LIN {X 0,Y 107.526,Z 478.473,A -85,B 0,C 180,E1 -28773.988,E2 -28773.988} C_VEL
LIN {X 0,Y 117.989,Z 469.59,A -85,B 0,C 180,E1 -28777.405,E2 -28777.405} C_VEL
LIN {X 0,Y 127.771,Z 459.826,A -85,B 0,C 180,E1 -28780.218,E2 -28780.218} C_VEL
LIN {X 0,Y 128.984,Z 458.465,A -85,B 0,C 180,E1 -28780.541,E2 -28780.541} C_VEL
LIN {X 0,Y 129.571,Z 457.629,A -85,B 0,C 180,E1 -28781.007,E2 -28781.007} C_VEL
LIN {X 0,Y 130.543,Z 454.991,A -85,B 0,C 180,E1 -28784.384,E2 -28784.384} C_VEL
LIN {X 0,Y 131.123,Z 453.011,A -85,B 0,C 180,E1 -28787.62,E2 -28787.62} C_VEL
LIN {X 0,Y 131.637,Z 451.555,A -85,B 0,C 180,E1 -28790.783,E2 -28790.783} C_VEL
LIN {X 0,Y 132.063,Z 450.596,A -85,B 0,C 180,E1 -28793.89,E2 -28793.89} C_VEL
LIN {X 0,Y 132.436,Z 450.06,A -85,B 0,C 180,E1 -28796.958,E2 -28796.958} C_VEL
LIN {X 0,Y 132.765,Z 450.031,A -85,B 0,C 180,E1 -28800,E2 -28800} C_VEL
LIN {X 0,Y 132.291,Z 452.688,A -85,B 0,C 180,E1 -28806.099,E2 -28806.099} C_VEL
LIN {X 0,Y 132.117,Z 455.556,A -85,B 0,C 180,E1 -28810.73,E2 -28810.73} C_VEL
LIN {X 0,Y 131.781,Z 457.018,A -85,B 0,C 180,E1 -28812.317,E2 -28812.317} C_VEL
LIN {X 0,Y 130.688,Z 459.886,A -85,B 0,C 180,E1 -28814.539,E2 -28814.539} C_VEL
LIN {X 0,Y 128.33,Z 462.983,A -85,B 0,C 180,E1 -28815.54,E2 -28815.54} C_VEL
LIN {X 0,Y 124.785,Z 467.253,A -85,B 0,C 180,E1 -28816.775,E2 -28816.775} C_VEL
LIN {X 0,Y 115.231,Z 476.64,A -85,B 0,C 180,E1 -28819.031,E2 -28819.031} C_VEL
LIN {X 0,Y 104.384,Z 485.862,A -85,B 0,C 180,E1 -28822.218,E2 -28822.218} C_VEL
LIN {X 0,Y 94.042,Z 493.562,A -85,B 0,C 180,E1 -28826.263,E2 -28826.263} C_VEL
LIN {X 0,Y 82.992,Z 500.795,A -85,B 0,C 180,E1 -28832.133,E2 -28832.133} C_VEL
LIN {X 0,Y 73.155,Z 506.533,A -85,B 0,C 180,E1 -28839.777,E2 -28839.777} C_VEL
LIN {X 0,Y 64.941,Z 510.906,A -85,B 0,C 180,E1 -28849.511,E2 -28849.511} C_VEL
LIN {X 0,Y 59.141,Z 514.04,A -85,B 0,C 180,E1 -28861.62,E2 -28861.62} C_VEL
LIN {X 0,Y 56.399,Z 515.993,A -85,B 0,C 180,E1 -28875.57,E2 -28875.57} C_VEL
LIN {X 0,Y 56.417,Z 516.621,A -85,B 0,C 180,E1 -28885.254,E2 -28885.254} C_VEL
LIN {X 0,Y 56.759,Z 516.763,A -85,B 0,C 180,E1 -28890.002,E2 -28890.002} C_VEL
LIN {X 0,Y 56.271,Z 516.528,A -85,B 0,C 180,E1 -28897.176,E2 -28897.176} C_VEL
LIN {X 0,Y 57.371,Z 515.135,A -85,B 0,C 180,E1 -28911.563,E2 -28911.563} C_VEL
LIN {X 0,Y 61.729,Z 512.574,A -85,B 0,C 180,E1 -28924.701,E2 -28924.701} C_VEL
LIN {X 0,Y 68.815,Z 508.797,A -85,B 0,C 180,E1 -28935.637,E2 -28935.637} C_VEL
LIN {X 0,Y 77.914,Z 503.726,A -85,B 0,C 180,E1 -28944.276,E2 -28944.276} C_VEL
LIN {X 0,Y 82.077,Z 501.289,A -85,B 0,C 180,E1 -28947.182,E2 -28947.182} C_VEL
LIN {X 0,Y 81.605,Z 500.684,A -85,B 0,C 180,E1 -28948.887,E2 -28948.887} C_VEL
LIN {X 0,Y 73.77,Z 497.104,A -85,B 0,C 180,E1 -28969.016,E2 -28969.016} C_VEL
LIN {X 0,Y 77.368,Z 492.97,A -85,B 0,C 180,E1 -28990.468,E2 -28990.468} C_VEL
LIN {X 0,Y 91.322,Z 488.038,A -85,B 0,C 180,E1 -29007.501,E2 -29007.501} C_VEL
LIN {X 0,Y 96.038,Z 486.659,A -85,B 0,C 180,E1 -29010.815,E2 -29010.815} C_VEL
LIN {X 0,Y 86.856,Z 492.48,A -85,B 0,C 180,E1 -29015.985,E2 -29015.985} C_VEL
LIN {X 0,Y 77.135,Z 497.86,A -85,B 0,C 180,E1 -29023.203,E2 -29023.203} C_VEL
LIN {X 0,Y 68.838,Z 501.906,A -85,B 0,C 180,E1 -29032.223,E2 -29032.223} C_VEL
LIN {X 0,Y 62.437,Z 504.726,A -85,B 0,C 180,E1 -29043.239,E2 -29043.239} C_VEL
LIN {X 0,Y 58.463,Z 506.395,A -85,B 0,C 180,E1 -29056.087,E2 -29056.087} C_VEL
LIN {X 0,Y 57.098,Z 506.97,A -85,B 0,C 180,E1 -29069.998,E2 -29069.998} C_VEL
LIN {X 0,Y 57.221,Z 506.877,A -85,B 0,C 180,E1 -29074.705,E2 -29074.705} C_VEL
LIN {X 0,Y 57.184,Z 506.725,A -85,B 0,C 180,E1 -29080.613,E2 -29080.613} C_VEL
LIN {X 0,Y 56.44,Z 506.175,A -85,B 0,C 180,E1 -29090.581,E2 -29090.581} C_VEL
LIN {X 0,Y 56.795,Z 505.428,A -85,B 0,C 180,E1 -29098.63,E2 -29098.63} C_VEL
LIN {X 0,Y 58.456,Z 504.577,A -85,B 0,C 180,E1 -29104.251,E2 -29104.251} C_VEL
LIN {X 0,Y 59.361,Z 504.195,A -85,B 0,C 180,E1 -29105.938,E2 -29105.938} C_VEL
LIN {X 0,Y 67.686,Z 500.765,A -85,B 0,C 180,E1 -29116.619,E2 -29116.619} C_VEL
LIN {X 0,Y 77.446,Z 496.115,A -85,B 0,C 180,E1 -29124.756,E2 -29124.756} C_VEL
LIN {X 0,Y 88.406,Z 490.04,A -85,B 0,C 180,E1 -29130.98,E2 -29130.98} C_VEL
LIN {X 0,Y 98.586,Z 483.468,A -85,B 0,C 180,E1 -29135.355,E2 -29135.355} C_VEL
LIN {X 0,Y 109.212,Z 475.482,A -85,B 0,C 180,E1 -29138.922,E2 -29138.922} C_VEL
LIN {X 0,Y 120.138,Z 465.853,A -85,B 0,C 180,E1 -29141.916,E2 -29141.916} C_VEL
LIN {X 0,Y 124.862,Z 461.121,A -85,B 0,C 180,E1 -29143.107,E2 -29143.107} C_VEL
LIN {X 0,Y 125.955,Z 458.558,A -85,B 0,C 180,E1 -29147.103,E2 -29147.103} C_VEL
LIN {X 0,Y 126.653,Z 457.034,A -85,B 0,C 180,E1 -29150.417,E2 -29150.417} C_VEL
LIN {X 0,Y 127.241,Z 455.957,A -85,B 0,C 180,E1 -29153.824,E2 -29153.824} C_VEL
LIN {X 0,Y 127.688,Z 455.429,A -85,B 0,C 180,E1 -29156.844,E2 -29156.844} C_VEL
LIN {X 0,Y 128.024,Z 455.44,A -85,B 0,C 180,E1 -29160,E2 -29160} C_VEL
LIN {X 0,Y 127.395,Z 458.175,A -85,B 0,C 180,E1 -29166.334,E2 -29166.334} C_VEL
LIN {X 0,Y 127.202,Z 460.04,A -85,B 0,C 180,E1 -29169.541,E2 -29169.541} C_VEL
LIN {X 0,Y 126.769,Z 461.429,A -85,B 0,C 180,E1 -29171.188,E2 -29171.188} C_VEL
LIN {X 0,Y 126.294,Z 462.429,A -85,B 0,C 180,E1 -29172.045,E2 -29172.045} C_VEL
LIN {X 0,Y 125.214,Z 463.892,A -85,B 0,C 180,E1 -29172.688,E2 -29172.688} C_VEL
LIN {X 0,Y 121.266,Z 468.283,A -85,B 0,C 180,E1 -29173.895,E2 -29173.895} C_VEL
LIN {X 0,Y 111.484,Z 477.437,A -85,B 0,C 180,E1 -29175.98,E2 -29175.98} C_VEL
LIN {X 0,Y 100.318,Z 486.437,A -85,B 0,C 180,E1 -29178.957,E2 -29178.957} C_VEL
LIN {X 0,Y 89.346,Z 494.125,A -85,B 0,C 180,E1 -29182.908,E2 -29182.908} C_VEL
LIN {X 0,Y 79.386,Z 500.177,A -85,B 0,C 180,E1 -29187.714,E2 -29187.714} C_VEL
LIN {X 0,Y 68.757,Z 505.913,A -85,B 0,C 180,E1 -29195.145,E2 -29195.145} C_VEL
LIN {X 0,Y 59.647,Z 510.288,A -85,B 0,C 180,E1 -29205.014,E2 -29205.014} C_VEL
LIN {X 0,Y 52.924,Z 513.422,A -85,B 0,C 180,E1 -29217.917,E2 -29217.917} C_VEL
LIN {X 0,Y 49.466,Z 515.374,A -85,B 0,C 180,E1 -29233.494,E2 -29233.494} C_VEL
LIN {X 0,Y 49.664,Z 516.153,A -85,B 0,C 180,E1 -29250.002,E2 -29250.002} C_VEL
LIN {X 0,Y 49.47,Z 515.358,A -85,B 0,C 180,E1 -29266.509,E2 -29266.509} C_VEL
LIN {X 0,Y 52.938,Z 513.383,A -85,B 0,C 180,E1 -29282.078,E2 -29282.078} C_VEL
LIN {X 0,Y 59.748,Z 510.176,A -85,B 0,C 180,E1 -29295.11,E2 -29295.11} C_VEL
LIN {X 0,Y 68.765,Z 505.809,A -85,B 0,C 180,E1 -29304.85,E2 -29304.85} C_VEL
LIN {X 0,Y 73.943,Z 503.107,A -85,B 0,C 180,E1 -29308.808,E2 -29308.808} C_VEL
LIN {X 0,Y 70.298,Z 501.756,A -85,B 0,C 180,E1 -29316.429,E2 -29316.429} C_VEL
LIN {X 0,Y 67.556,Z 498.082,A -85,B 0,C 180,E1 -29340.001,E2 -29340.001} C_VEL
LIN {X 0,Y 77.122,Z 493.753,A -85,B 0,C 180,E1 -29361.378,E2 -29361.378} C_VEL
LIN {X 0,Y 85.588,Z 491.331,A -85,B 0,C 180,E1 -29369.518,E2 -29369.518} C_VEL
LIN {X 0,Y 82.898,Z 493.088,A -85,B 0,C 180,E1 -29372.025,E2 -29372.025} C_VEL
LIN {X 0,Y 72.47,Z 498.469,A -85,B 0,C 180,E1 -29379.118,E2 -29379.118} C_VEL
LIN {X 0,Y 63.395,Z 502.514,A -85,B 0,C 180,E1 -29388.303,E2 -29388.303} C_VEL
LIN {X 0,Y 56.21,Z 505.335,A -85,B 0,C 180,E1 -29399.99,E2 -29399.99} C_VEL
LIN {X 0,Y 51.637,Z 507.003,A -85,B 0,C 180,E1 -29414.203,E2 -29414.203} C_VEL
LIN {X 0,Y 50.034,Z 507.577,A -85,B 0,C 180,E1 -29429.998,E2 -29429.998} C_VEL
LIN {X 0,Y 51.628,Z 507.025,A -85,B 0,C 180,E1 -29445.797,E2 -29445.797} C_VEL
LIN {X 0,Y 56.208,Z 505.386,A -85,B 0,C 180,E1 -29460.008,E2 -29460.008} C_VEL
LIN {X 0,Y 59.361,Z 504.195,A -85,B 0,C 180,E1 -29465.938,E2 -29465.938} C_VEL
LIN {X 0,Y 61.922,Z 503.134,A -85,B 0,C 180,E1 -29470.878,E2 -29470.878} C_VEL
LIN {X 0,Y 65.425,Z 501.144,A -85,B 0,C 180,E1 -29479.068,E2 -29479.068} C_VEL
LIN {X 0,Y 69.953,Z 498.569,A -85,B 0,C 180,E1 -29486.246,E2 -29486.246} C_VEL
LIN {X 0,Y 73.849,Z 496.592,A -85,B 0,C 180,E1 -29489.427,E2 -29489.427} C_VEL
LIN {X 0,Y 85.193,Z 490.646,A -85,B 0,C 180,E1 -29495.153,E2 -29495.153} C_VEL
LIN {X 0,Y 95.842,Z 484.074,A -85,B 0,C 180,E1 -29499.217,E2 -29499.217} C_VEL
LIN {X 0,Y 106.868,Z 476.086,A -85,B 0,C 180,E1 -29502.47,E2 -29502.47} C_VEL
LIN {X 0,Y 117.696,Z 466.844,A -85,B 0,C 180,E1 -29505.092,E2 -29505.092} C_VEL
LIN {X 0,Y 118.875,Z 465.741,A -85,B 0,C 180,E1 -29505.372,E2 -29505.372} C_VEL
LIN {X 0,Y 120.504,Z 463.923,A -85,B 0,C 180,E1 -29506.509,E2 -29506.509} C_VEL
LIN {X 0,Y 121.393,Z 462.343,A -85,B 0,C 180,E1 -29509.998,E2 -29509.998} C_VEL
LIN {X 0,Y 122.106,Z 461.238,A -85,B 0,C 180,E1 -29513.389,E2 -29513.389} C_VEL
LIN {X 0,Y 122.724,Z 460.598,A -85,B 0,C 180,E1 -29516.717,E2 -29516.717} C_VEL
LIN {X 0,Y 123.049,Z 460.665,A -85,B 0,C 180,E1 -29520,E2 -29520} C_VEL
LIN {X 0,Y 122.599,Z 461.915,A -85,B 0,C 180,E1 -29523.286,E2 -29523.286} C_VEL
LIN {X 0,Y 122.105,Z 464.378,A -85,B 0,C 180,E1 -29528.273,E2 -29528.273} C_VEL
LIN {X 0,Y 121.328,Z 465.99,A -85,B 0,C 180,E1 -29530.026,E2 -29530.026} C_VEL
LIN {X 0,Y 118.069,Z 469.312,A -85,B 0,C 180,E1 -29530.844,E2 -29530.844} C_VEL
LIN {X 0,Y 106.405,Z 479.555,A -85,B 0,C 180,E1 -29533.039,E2 -29533.039} C_VEL
LIN {X 0,Y 94.989,Z 488.091,A -85,B 0,C 180,E1 -29535.883,E2 -29535.883} C_VEL
LIN {X 0,Y 82.372,Z 496.143,A -85,B 0,C 180,E1 -29540.199,E2 -29540.199} C_VEL
LIN {X 0,Y 70.458,Z 502.606,A -85,B 0,C 180,E1 -29546.142,E2 -29546.142} C_VEL
LIN {X 0,Y 59.64,Z 507.648,A -85,B 0,C 180,E1 -29554.426,E2 -29554.426} C_VEL
LIN {X 0,Y 50.527,Z 511.386,A -85,B 0,C 180,E1 -29565.938,E2 -29565.938} C_VEL
LIN {X 0,Y 44.306,Z 513.926,A -85,B 0,C 180,E1 -29581.586,E2 -29581.586} C_VEL
LIN {X 0,Y 42.068,Z 515.299,A -85,B 0,C 180,E1 -29600.385,E2 -29600.385} C_VEL
LIN {X 0,Y 42.54,Z 515.54,A -85,B 0,C 180,E1 -29610.002,E2 -29610.002} C_VEL
LIN {X 0,Y 42.644,Z 514.741,A -85,B 0,C 180,E1 -29629.247,E2 -29629.247} C_VEL
LIN {X 0,Y 47.003,Z 512.764,A -85,B 0,C 180,E1 -29646.735,E2 -29646.735} C_VEL
LIN {X 0,Y 54.795,Z 509.598,A -85,B 0,C 180,E1 -29660.317,E2 -29660.317} C_VEL
LIN {X 0,Y 64.885,Z 505.189,A -85,B 0,C 180,E1 -29670.06,E2 -29670.06} C_VEL
LIN {X 0,Y 64.229,Z 504.286,A -85,B 0,C 180,E1 -29674.045,E2 -29674.045} C_VEL
LIN {X 0,Y 60.89,Z 500.758,A -85,B 0,C 180,E1 -29700.001,E2 -29700.001} C_VEL
LIN {X 0,Y 70.968,Z 496.627,A -85,B 0,C 180,E1 -29723.337,E2 -29723.337} C_VEL
LIN {X 0,Y 75.912,Z 495.32,A -85,B 0,C 180,E1 -29728.589,E2 -29728.589} C_VEL
LIN {X 0,Y 74.908,Z 495.948,A -85,B 0,C 180,E1 -29730.05,E2 -29730.05} C_VEL
LIN {X 0,Y 63.066,Z 501.261,A -85,B 0,C 180,E1 -29738.731,E2 -29738.731} C_VEL
LIN {X 0,Y 53.96,Z 504.683,A -85,B 0,C 180,E1 -29749.364,E2 -29749.364} C_VEL
LIN {X 0,Y 47.165,Z 506.915,A -85,B 0,C 180,E1 -29763.444,E2 -29763.444} C_VEL
LIN {X 0,Y 43.45,Z 508.037,A -85,B 0,C 180,E1 -29780.689,E2 -29780.689} C_VEL
LIN {X 0,Y 43.441,Z 508.045,A -85,B 0,C 180,E1 -29799.308,E2 -29799.308} C_VEL
LIN {X 0,Y 47.305,Z 506.912,A -85,B 0,C 180,E1 -29816.948,E2 -29816.948} C_VEL
LIN {X 0,Y 53.952,Z 504.751,A -85,B 0,C 180,E1 -29830.639,E2 -29830.639} C_VEL
LIN {X 0,Y 63.033,Z 501.372,A -85,B 0,C 180,E1 -29841.302,E2 -29841.302} C_VEL
LIN {X 0,Y 73.849,Z 496.592,A -85,B 0,C 180,E1 -29849.427,E2 -29849.427} C_VEL
LIN {X 0,Y 77.902,Z 494.517,A -85,B 0,C 180,E1 -29852.256,E2 -29852.256} C_VEL
LIN {X 0,Y 83.796,Z 490.995,A -85,B 0,C 180,E1 -29857.353,E2 -29857.353} C_VEL
LIN {X 0,Y 90.008,Z 487.028,A -85,B 0,C 180,E1 -29861.739,E2 -29861.739} C_VEL
LIN {X 0,Y 94.336,Z 484.159,A -85,B 0,C 180,E1 -29863.49,E2 -29863.49} C_VEL
LIN {X 0,Y 106.611,Z 475.39,A -85,B 0,C 180,E1 -29866.491,E2 -29866.491} C_VEL
LIN {X 0,Y 114.862,Z 468.506,A -85,B 0,C 180,E1 -29868.23,E2 -29868.23} C_VEL
LIN {X 0,Y 115.819,Z 467.5,A -85,B 0,C 180,E1 -29869.511,E2 -29869.511} C_VEL
LIN {X 0,Y 116.751,Z 466.288,A -85,B 0,C 180,E1 -29873.085,E2 -29873.085} C_VEL
LIN {X 0,Y 117.521,Z 465.59,A -85,B 0,C 180,E1 -29876.571,E2 -29876.571} C_VEL
LIN {X 0,Y 117.868,Z 465.674,A -85,B 0,C 180,E1 -29880,E2 -29880} C_VEL
LIN {X 0,Y 116.903,Z 468.533,A -85,B 0,C 180,E1 -29886.905,E2 -29886.905} C_VEL
LIN {X 0,Y 115.039,Z 470.483,A -85,B 0,C 180,E1 -29887.651,E2 -29887.651} C_VEL
LIN {X 0,Y 103.328,Z 480.287,A -85,B 0,C 180,E1 -29889.521,E2 -29889.521} C_VEL
LIN {X 0,Y 91.621,Z 488.611,A -85,B 0,C 180,E1 -29892.041,E2 -29892.041} C_VEL
LIN {X 0,Y 80.177,Z 495.528,A -85,B 0,C 180,E1 -29895.377,E2 -29895.377} C_VEL
LIN {X 0,Y 67.595,Z 501.988,A -85,B 0,C 180,E1 -29900.654,E2 -29900.654} C_VEL
LIN {X 0,Y 55.886,Z 507.03,A -85,B 0,C 180,E1 -29908.325,E2 -29908.325} C_VEL
LIN {X 0,Y 45.632,Z 510.768,A -85,B 0,C 180,E1 -29919.642,E2 -29919.642} C_VEL
LIN {X 0,Y 38.114,Z 513.306,A -85,B 0,C 180,E1 -29936.417,E2 -29936.417} C_VEL
LIN {X 0,Y 35.028,Z 514.683,A -85,B 0,C 180,E1 -29958.428,E2 -29958.428} C_VEL
LIN {X 0,Y 35.417,Z 514.927,A -85,B 0,C 180,E1 -29970.003,E2 -29970.003} C_VEL
LIN {X 0,Y 35.932,Z 514.122,A -85,B 0,C 180,E1 -29993.031,E2 -29993.031} C_VEL
LIN {X 0,Y 41.448,Z 512.144,A -85,B 0,C 180,E1 -30012.709,E2 -30012.709} C_VEL
LIN {X 0,Y 50.504,Z 508.979,A -85,B 0,C 180,E1 -30026.613,E2 -30026.613} C_VEL
LIN {X 0,Y 55.889,Z 506.938,A -85,B 0,C 180,E1 -30031.676,E2 -30031.676} C_VEL
LIN {X 0,Y 57.087,Z 506.204,A -85,B 0,C 180,E1 -30033.851,E2 -30033.851} C_VEL
LIN {X 0,Y 54.104,Z 503.148,A -85,B 0,C 180,E1 -30060.001,E2 -30060.001} C_VEL
LIN {X 0,Y 65.838,Z 498.97,A -85,B 0,C 180,E1 -30086.934,E2 -30086.934} C_VEL
LIN {X 0,Y 64.464,Z 499.69,A -85,B 0,C 180,E1 -30089.285,E2 -30089.285} C_VEL
LIN {X 0,Y 53.641,Z 503.735,A -85,B 0,C 180,E1 -30098.173,E2 -30098.173} C_VEL
LIN {X 0,Y 44.51,Z 506.554,A -85,B 0,C 180,E1 -30110.829,E2 -30110.829} C_VEL
LIN {X 0,Y 38.245,Z 508.217,A -85,B 0,C 180,E1 -30128.434,E2 -30128.434} C_VEL
LIN {X 0,Y 35.912,Z 508.792,A -85,B 0,C 180,E1 -30149.997,E2 -30149.997} C_VEL
LIN {X 0,Y 38.237,Z 508.239,A -85,B 0,C 180,E1 -30171.565,E2 -30171.565} C_VEL
LIN {X 0,Y 44.507,Z 506.604,A -85,B 0,C 180,E1 -30189.168,E2 -30189.168} C_VEL
LIN {X 0,Y 53.614,Z 503.823,A -85,B 0,C 180,E1 -30201.858,E2 -30201.858} C_VEL
LIN {X 0,Y 64.427,Z 499.821,A -85,B 0,C 180,E1 -30210.768,E2 -30210.768} C_VEL
LIN {X 0,Y 73.248,Z 495.947,A -85,B 0,C 180,E1 -30215.711,E2 -30215.711} C_VEL
LIN {X 0,Y 85.802,Z 489.38,A -85,B 0,C 180,E1 -30220.874,E2 -30220.874} C_VEL
LIN {X 0,Y 94.336,Z 484.159,A -85,B 0,C 180,E1 -30223.49,E2 -30223.49} C_VEL
LIN {X 0,Y 97.161,Z 482.211,A -85,B 0,C 180,E1 -30224.686,E2 -30224.686} C_VEL
LIN {X 0,Y 105.078,Z 476.123,A -85,B 0,C 180,E1 -30229.839,E2 -30229.839} C_VEL
LIN {X 0,Y 107.938,Z 473.839,A -85,B 0,C 180,E1 -30230.724,E2 -30230.724} C_VEL
LIN {X 0,Y 109.627,Z 472.519,A -85,B 0,C 180,E1 -30231.011,E2 -30231.011} C_VEL
LIN {X 0,Y 111.137,Z 471.15,A -85,B 0,C 180,E1 -30232.734,E2 -30232.734} C_VEL
LIN {X 0,Y 112.083,Z 470.39,A -85,B 0,C 180,E1 -30236.405,E2 -30236.405} C_VEL
LIN {X 0,Y 112.447,Z 470.511,A -85,B 0,C 180,E1 -30240.081,E2 -30240.081} C_VEL
LIN {X 0,Y 111.822,Z 471.804,A -85,B 0,C 180,E1 -30243.603,E2 -30243.603} C_VEL
LIN {X 0,Y 110.058,Z 473.546,A -85,B 0,C 180,E1 -30244.589,E2 -30244.589} C_VEL
LIN {X 0,Y 97.226,Z 483.409,A -85,B 0,C 180,E1 -30246.329,E2 -30246.329} C_VEL
LIN {X 0,Y 85.304,Z 491.1,A -85,B 0,C 180,E1 -30248.645,E2 -30248.645} C_VEL
LIN {X 0,Y 71.927,Z 498.326,A -85,B 0,C 180,E1 -30252.291,E2 -30252.291} C_VEL
LIN {X 0,Y 59.017,Z 504.058,A -85,B 0,C 180,E1 -30257.702,E2 -30257.702} C_VEL
LIN {X 0,Y 46.933,Z 508.436,A -85,B 0,C 180,E1 -30266.045,E2 -30266.045} C_VEL
LIN {X 0,Y 36.464,Z 511.564,A -85,B 0,C 180,E1 -30279.564,E2 -30279.564} C_VEL
LIN {X 0,Y 29.455,Z 513.522,A -85,B 0,C 180,E1 -30301.5,E2 -30301.5} C_VEL
LIN {X 0,Y 28.289,Z 514.314,A -85,B 0,C 180,E1 -30330.003,E2 -30330.003} C_VEL
LIN {X 0,Y 29.461,Z 513.505,A -85,B 0,C 180,E1 -30358.5,E2 -30358.5} C_VEL
LIN {X 0,Y 36.486,Z 511.524,A -85,B 0,C 180,E1 -30380.402,E2 -30380.402} C_VEL
LIN {X 0,Y 46.936,Z 508.361,A -85,B 0,C 180,E1 -30393.956,E2 -30393.956} C_VEL
LIN {X 0,Y 48.854,Z 507.498,A -85,B 0,C 180,E1 -30397.152,E2 -30397.152} C_VEL
LIN {X 0,Y 48.703,Z 504.355,A -85,B 0,C 180,E1 -30428.298,E2 -30428.298} C_VEL
LIN {X 0,Y 56.342,Z 502.07,A -85,B 0,C 180,E1 -30445.491,E2 -30445.491} C_VEL
LIN {X 0,Y 55.323,Z 502.479,A -85,B 0,C 180,E1 -30447.217,E2 -30447.217} C_VEL
LIN {X 0,Y 44.192,Z 505.901,A -85,B 0,C 180,E1 -30457.326,E2 -30457.326} C_VEL
LIN {X 0,Y 34.44,Z 508.26,A -85,B 0,C 180,E1 -30474.715,E2 -30474.715} C_VEL
LIN {X 0,Y 29.605,Z 509.252,A -85,B 0,C 180,E1 -30496.264,E2 -30496.264} C_VEL
LIN {X 0,Y 29.596,Z 509.259,A -85,B 0,C 180,E1 -30523.734,E2 -30523.734} C_VEL
LIN {X 0,Y 35.068,Z 508.168,A -85,B 0,C 180,E1 -30546.955,E2 -30546.955} C_VEL
LIN {X 0,Y 44.183,Z 505.967,A -85,B 0,C 180,E1 -30562.683,E2 -30562.683} C_VEL
LIN {X 0,Y 55.291,Z 502.589,A -85,B 0,C 180,E1 -30572.841,E2 -30572.841} C_VEL
LIN {X 0,Y 67.447,Z 497.938,A -85,B 0,C 180,E1 -30579.682,E2 -30579.682} C_VEL
LIN {X 0,Y 77.036,Z 493.518,A -85,B 0,C 180,E1 -30583.315,E2 -30583.315} C_VEL
LIN {X 0,Y 90.12,Z 486.284,A -85,B 0,C 180,E1 -30587.109,E2 -30587.109} C_VEL
LIN {X 0,Y 103.488,Z 477.293,A -85,B 0,C 180,E1 -30589.963,E2 -30589.963} C_VEL
LIN {X 0,Y 107.938,Z 473.839,A -85,B 0,C 180,E1 -30590.724,E2 -30590.724} C_VEL
LIN {X 0,Y 108.721,Z 473.199,A -85,B 0,C 180,E1 -30591.295,E2 -30591.295} C_VEL
LIN {X 0,Y 108.87,Z 473.035,A -85,B 0,C 180,E1 -30592.392,E2 -30592.392} C_VEL
LIN {X 0,Y 108.419,Z 473.362,A -85,B 0,C 180,E1 -30593.687,E2 -30593.687} C_VEL
LIN {X 0,Y 106.621,Z 474.912,A -85,B 0,C 180,E1 -30597.309,E2 -30597.309} C_VEL
LIN {X 0,Y 106.589,Z 475.027,A -85,B 0,C 180,E1 -30598.189,E2 -30598.189} C_VEL
LIN {X 0,Y 106.857,Z 475.068,A -85,B 0,C 180,E1 -30600,E2 -30600} C_VEL
LIN {X 0,Y 105.443,Z 476.362,A -85,B 0,C 180,E1 -30601.243,E2 -30601.243} C_VEL
LIN {X 0,Y 93.211,Z 485.116,A -85,B 0,C 180,E1 -30602.537,E2 -30602.537} C_VEL
LIN {X 0,Y 81.063,Z 492.446,A -85,B 0,C 180,E1 -30604.429,E2 -30604.429} C_VEL
LIN {X 0,Y 67.334,Z 499.278,A -85,B 0,C 180,E1 -30607.458,E2 -30607.458} C_VEL
LIN {X 0,Y 53.927,Z 504.674,A -85,B 0,C 180,E1 -30612.204,E2 -30612.204} C_VEL
LIN {X 0,Y 41.101,Z 508.757,A -85,B 0,C 180,E1 -30619.997,E2 -30619.997} C_VEL
LIN {X 0,Y 32.365,Z 510.947,A -85,B 0,C 180,E1 -30629.709,E2 -30629.709} C_VEL
LIN {X 0,Y 23.38,Z 512.903,A -85,B 0,C 180,E1 -30653.048,E2 -30653.048} C_VEL
LIN {X 0,Y 21.172,Z 513.702,A -85,B 0,C 180,E1 -30690.004,E2 -30690.004} C_VEL
LIN {X 0,Y 23.388,Z 512.885,A -85,B 0,C 180,E1 -30726.947,E2 -30726.947} C_VEL
LIN {X 0,Y 32.38,Z 510.905,A -85,B 0,C 180,E1 -30750.255,E2 -30750.255} C_VEL
LIN {X 0,Y 41.062,Z 508.701,A -85,B 0,C 180,E1 -30759.983,E2 -30759.983} C_VEL
LIN {X 0,Y 44.573,Z 505.345,A -85,B 0,C 180,E1 -30798.383,E2 -30798.383} C_VEL
LIN {X 0,Y 46.253,Z 504.953,A -85,B 0,C 180,E1 -30804.255,E2 -30804.255} C_VEL
LIN {X 0,Y 34.705,Z 507.772,A -85,B 0,C 180,E1 -30815.897,E2 -30815.897} C_VEL
LIN {X 0,Y 25.645,Z 509.432,A -85,B 0,C 180,E1 -30836.759,E2 -30836.759} C_VEL
LIN {X 0,Y 21.794,Z 510.006,A -85,B 0,C 180,E1 -30869.996,E2 -30869.996} C_VEL
LIN {X 0,Y 25.638,Z 509.453,A -85,B 0,C 180,E1 -30903.243,E2 -30903.243} C_VEL
LIN {X 0,Y 34.701,Z 507.82,A -85,B 0,C 180,E1 -30924.103,E2 -30924.103} C_VEL
LIN {X 0,Y 46.23,Z 505.039,A -85,B 0,C 180,E1 -30935.798,E2 -30935.798} C_VEL
LIN {X 0,Y 58.821,Z 501.036,A -85,B 0,C 180,E1 -30942.905,E2 -30942.905} C_VEL
LIN {X 0,Y 68.65,Z 497.16,A -85,B 0,C 180,E1 -30946.542,E2 -30946.542} C_VEL
LIN {X 0,Y 83.412,Z 489.99,A -85,B 0,C 180,E1 -30950.493,E2 -30950.493} C_VEL
LIN {X 0,Y 95.635,Z 482.629,A -85,B 0,C 180,E1 -30952.781,E2 -30952.781} C_VEL
LIN {X 0,Y 105.481,Z 475.627,A -85,B 0,C 180,E1 -30954.347,E2 -30954.347} C_VEL
LIN {X 0,Y 105.912,Z 475.299,A -85,B 0,C 180,E1 -30954.47,E2 -30954.47} C_VEL
LIN {X 0,Y 106.419,Z 474.982,A -85,B 0,C 180,E1 -30956.213,E2 -30956.213} C_VEL
LIN {X 0,Y 106.589,Z 475.027,A -85,B 0,C 180,E1 -30958.189,E2 -30958.189} C_VEL
LIN {X 0,Y 106.03,Z 475.559,A -85,B 0,C 180,E1 -30958.994,E2 -30958.994} C_VEL
LIN {X 0,Y 104.37,Z 476.906,A -85,B 0,C 180,E1 -30959.582,E2 -30959.582} C_VEL
LIN {X 0,Y 101.332,Z 479.192,A -85,B 0,C 180,E1 -30959.75,E2 -30959.75} C_VEL
LIN {X 0,Y 91.572,Z 485.593,A -85,B 0,C 180,E1 -30958.449,E2 -30958.449} C_VEL
LIN {X 0,Y 89.058,Z 487.114,A -85,B 0,C 180,E1 -30958.48,E2 -30958.48} C_VEL
LIN {X 0,Y 74.152,Z 495.267,A -85,B 0,C 180,E1 -30960.176,E2 -30960.176} C_VEL
LIN {X 0,Y 59.805,Z 501.53,A -85,B 0,C 180,E1 -30962.736,E2 -30962.736} C_VEL
LIN {X 0,Y 46.015,Z 506.254,A -85,B 0,C 180,E1 -30966.91,E2 -30966.91} C_VEL
LIN {X 0,Y 35.932,Z 508.913,A -85,B 0,C 180,E1 -30972.065,E2 -30972.065} C_VEL
LIN {X 0,Y 23.387,Z 511.447,A -85,B 0,C 180,E1 -30985.649,E2 -30985.649} C_VEL
LIN {X 0,Y 14.573,Z 512.83,A -85,B 0,C 180,E1 -31021.174,E2 -31021.174} C_VEL
LIN {X 0,Y 14.012,Z 513.086,A -85,B 0,C 180,E1 -31050.006,E2 -31050.006} C_VEL
LIN {X 0,Y 18.166,Z 512.267,A -85,B 0,C 180,E1 -31100.699,E2 -31100.699} C_VEL
LIN {X 0,Y 29.476,Z 510.285,A -85,B 0,C 180,E1 -31122.509,E2 -31122.509} C_VEL
LIN {X 0,Y 33.173,Z 509.371,A -85,B 0,C 180,E1 -31127.77,E2 -31127.77} C_VEL
LIN {X 0,Y 36.743,Z 507.268,A -85,B 0,C 180,E1 -31158.213,E2 -31158.213} C_VEL
LIN {X 0,Y 35.451,Z 507.533,A -85,B 0,C 180,E1 -31161.208,E2 -31161.208} C_VEL
LIN {X 0,Y 23.27,Z 509.622,A -85,B 0,C 180,E1 -31177.161,E2 -31177.161} C_VEL
LIN {X 0,Y 16.244,Z 510.466,A -85,B 0,C 180,E1 -31204.357,E2 -31204.357} C_VEL
LIN {X 0,Y 16.235,Z 510.473,A -85,B 0,C 180,E1 -31255.644,E2 -31255.644} C_VEL
LIN {X 0,Y 25.245,Z 509.383,A -85,B 0,C 180,E1 -31286.629,E2 -31286.629} C_VEL
LIN {X 0,Y 37.334,Z 507.184,A -85,B 0,C 180,E1 -31300.252,E2 -31300.252} C_VEL
LIN {X 0,Y 50.419,Z 503.806,A -85,B 0,C 180,E1 -31307.345,E2 -31307.345} C_VEL
LIN {X 0,Y 63.925,Z 499.151,A -85,B 0,C 180,E1 -31311.672,E2 -31311.672} C_VEL
LIN {X 0,Y 74.218,Z 494.732,A -85,B 0,C 180,E1 -31313.865,E2 -31313.865} C_VEL
LIN {X 0,Y 88.049,Z 487.495,A -85,B 0,C 180,E1 -31316.137,E2 -31316.137} C_VEL
LIN {X 0,Y 98.488,Z 480.899,A -85,B 0,C 180,E1 -31317.445,E2 -31317.445} C_VEL
LIN {X 0,Y 98.467,Z 480.943,A -85,B 0,C 180,E1 -31317.74,E2 -31317.74} C_VEL
LIN {X 0,Y 89.058,Z 487.114,A -85,B 0,C 180,E1 -31318.48,E2 -31318.48} C_VEL
LIN {X 0,Y 88.082,Z 488.838,A -85,B 0,C 180,E1 -31318.567,E2 -31318.567} C_VEL
LIN {X 0,Y 88.082,Z 514.711,A -85,B 0,C 180,E1 -31318.567,E2 -31318.567} C_VEL
LIN {X 0,Y 51.515,Z 514.711,A -85,B 0,C 180,E1 -31313.509,E2 -31313.509} C_VEL
LIN {X 0,Y 49.561,Z 512.711,A -85,B 0,C 180,E1 -31313.024,E2 -31313.024} C_VEL
LIN {X 0,Y 49.561,Z 506.417,A -85,B 0,C 180,E1 -31313.024,E2 -31313.024} C_VEL
LIN {X 0,Y 49.345,Z 504.424,A -85,B 0,C 180,E1 -31315.527,E2 -31315.527} C_VEL
LIN {X 0,Y 49.251,Z 504.552,A -85,B 0,C 180,E1 -31317.26,E2 -31317.26} C_VEL
LIN {X 0,Y 35.14,Z 508.293,A -85,B 0,C 180,E1 -31320.477,E2 -31320.477} C_VEL
LIN {X 0,Y 21.283,Z 510.827,A -85,B 0,C 180,E1 -31327.88,E2 -31327.88} C_VEL
LIN {X 0,Y 8.975,Z 512.212,A -85,B 0,C 180,E1 -31358.474,E2 -31358.474} C_VEL
LIN {X 0,Y 6.826,Z 512.468,A -85,B 0,C 180,E1 -31410.013,E2 -31410.013} C_VEL
LIN {X 0,Y 14.698,Z 511.646,A -85,B 0,C 180,E1 -31483.029,E2 -31483.029} C_VEL
LIN {X 0,Y 25.044,Z 510.219,A -85,B 0,C 180,E1 -31494.88,E2 -31494.88} C_VEL
LIN {X 0,Y 26.231,Z 509.822,A -85,B 0,C 180,E1 -31500.002,E2 -31500.002} C_VEL
LIN {X 0,Y 27.359,Z 509.287,A -85,B 0,C 180,E1 -31510.494,E2 -31510.494} C_VEL
LIN {X 0,Y 24.767,Z 509.631,A -85,B 0,C 180,E1 -31515.363,E2 -31515.363} C_VEL
LIN {X 0,Y 15.842,Z 510.649,A -85,B 0,C 180,E1 -31527.457,E2 -31527.457} C_VEL
LIN {X 0,Y 7.682,Z 511.22,A -85,B 0,C 180,E1 -31589.988,E2 -31589.988} C_VEL
LIN {X 0,Y 15.837,Z 510.669,A -85,B 0,C 180,E1 -31652.553,E2 -31652.553} C_VEL
LIN {X 0,Y 28.782,Z 509.037,A -85,B 0,C 180,E1 -31667.597,E2 -31667.597} C_VEL
LIN {X 0,Y 42.434,Z 506.258,A -85,B 0,C 180,E1 -31673.563,E2 -31673.563} C_VEL
LIN {X 0,Y 49.345,Z 504.424,A -85,B 0,C 180,E1 -31675.527,E2 -31675.527} C_VEL
LIN {X 0,Y 49.229,Z 506.424,A -85,B 0,C 180,E1 -31677.849,E2 -31677.849} C_VEL
LIN {X 0,Y 49.229,Z 600,A -85,B 0,C 180,E1 -31677.849,E2 -31677.849} C_VEL
LIN {X 0,Y 49.229,Z 600,A -85,B 0,C 180,E1 -31677.849,E2 -31677.849}

QRS_NEXT_CUT()

QRS_NEXT()
QRS_HOME()

END
